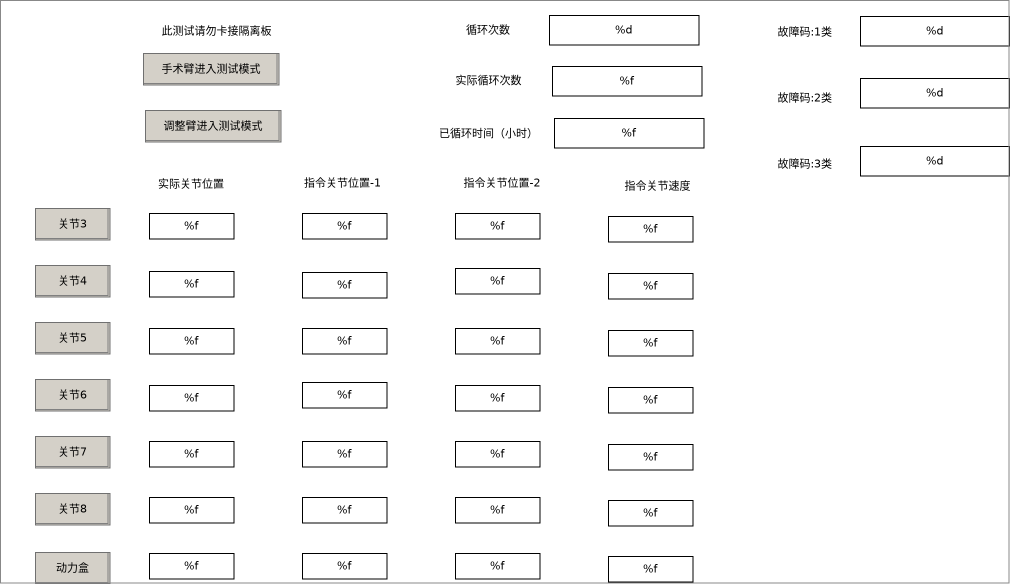
VISUALIZATION arm4CycleTest  // 1010x584
VAR_IN_OUT
	
END_VAR
VAR CONSTANT
	arm : INT := 4;
END_VAR
    Button (143,53 136x32), "手术臂进入测试模式", colour toggle: g_cycleTest.m_enterCycleTestMode[4]
        toggle g_cycleTest.m_enterCycleTestMode[4]
    Rectangle (549,15 150x30), "%d", text variable: g_cycleTest.m_targetCycleNum[4]
    Label (446,15 84x30), "循环次数"
    Label (283,169 119x28), "指令关节位置-1"
    Label (141,169 100x30), "实际关节位置"
    Rectangle (149,385 85x26), "%f", text variable: g_systemInfo.m_slaveJntInfo[4,1].m_curJntPos
    Rectangle (149,441 85x26), "%f", text variable: g_systemInfo.m_slaveJntInfo[4,2].m_curJntPos
    Rectangle (149,497 85x26), "%f", text variable: g_systemInfo.m_slaveJntInfo[4,3].m_curJntPos
    Rectangle (149,553 85x26), "%f", text variable: g_systemInfo.m_slaveJntInfo[4,4].m_curJntPos
    Rectangle (149,213 85x26), "%f", text variable: g_systemInfo.m_setupJntInfo[4,3].m_curJntPos
    Rectangle (149,271 85x26), "%f", text variable: g_systemInfo.m_setupJntInfo[4,4].m_curJntPos
    Rectangle (149,328 85x26), "%f", text variable: g_systemInfo.m_setupJntInfo[4,5].m_curJntPos
    Rectangle (302,213 85x26), "%f", text variable: g_cycleTest.m_targetJntPosSetup[4,1][3]
        OnMouseClick: write the text variable via Default
    Rectangle (302,272 85x26), "%f", text variable: g_cycleTest.m_targetJntPosSetup[4,1][4]
        OnMouseClick: write the text variable via Default
    Rectangle (302,328 85x26), "%f", text variable: g_cycleTest.m_targetJntPosSetup[4,1][5]
        OnMouseClick: write the text variable via Default
    Rectangle (302,382 85x26), "%f", text variable: g_cycleTest.m_targetJntPos[4,1][1]
        OnMouseClick: write the text variable via Default
    Rectangle (302,441 85x26), "%f", text variable: g_cycleTest.m_targetJntPos[4,1][2]
        OnMouseClick: write the text variable via Default
    Rectangle (302,497 85x26), "%f", text variable: g_cycleTest.m_targetJntPos[4,1][3]
        OnMouseClick: write the text variable via Default
    Rectangle (302,553 85x26), "%f", text variable: g_cycleTest.m_targetJntPos[4,1][4]
        OnMouseClick: write the text variable via Default
    Label (444,169 116x28), "指令关节位置-2"
    Rectangle (455,213 85x26), "%f", text variable: g_cycleTest.m_targetJntPosSetup[4,2][3]
        OnMouseClick: write the text variable via Default
    Rectangle (455,268 85x26), "%f", text variable: g_cycleTest.m_targetJntPosSetup[4,2][4]
        OnMouseClick: write the text variable via Default
    Rectangle (455,328 85x26), "%f", text variable: g_cycleTest.m_targetJntPosSetup[4,2][5]
        OnMouseClick: write the text variable via Default
    Rectangle (455,385 85x26), "%f", text variable: g_cycleTest.m_targetJntPos[4,2][1]
        OnMouseClick: write the text variable via Default
    Rectangle (455,441 85x26), "%f", text variable: g_cycleTest.m_targetJntPos[4,2][2]
        OnMouseClick: write the text variable via Default
    Rectangle (455,497 85x26), "%f", text variable: g_cycleTest.m_targetJntPos[4,2][3]
        OnMouseClick: write the text variable via Default
    Rectangle (455,553 85x26), "%f", text variable: g_cycleTest.m_targetJntPos[4,2][4]
        OnMouseClick: write the text variable via Default
    Button (145,110 136x32), "调整臂进入测试模式", colour toggle: g_cycleTest.m_enterCycleTestModeSetup[4]
        toggle g_cycleTest.m_enterCycleTestModeSetup[4]
    Label (603,172 109x28), "指令关节速度"
    Rectangle (608,216 85x26), "%f", text variable: g_cycleTest.m_targetJntVelSetup[4][3]
        OnMouseClick: write the text variable via Default
    Rectangle (608,273 85x26), "%f", text variable: g_cycleTest.m_targetJntVelSetup[4][4]
        OnMouseClick: write the text variable via Default
    Rectangle (608,330 85x26), "%f", text variable: g_cycleTest.m_targetJntVelSetup[4][5]
        OnMouseClick: write the text variable via Default
    Rectangle (608,387 85x26), "%f", text variable: g_cycleTest.m_targetJntVelSlave[4][1]
        OnMouseClick: write the text variable via Default
    Rectangle (608,444 85x26), "%f", text variable: g_cycleTest.m_targetJntVelSlave[4][2]
        OnMouseClick: write the text variable via Default
    Rectangle (608,500 85x26), "%f", text variable: g_cycleTest.m_targetJntVelSlave[4][3]
        OnMouseClick: write the text variable via Default
    Rectangle (608,556 85x26), "%f", text variable: g_cycleTest.m_targetJntVelSlave[4][4]
        OnMouseClick: write the text variable via Default
    Rectangle (552,66 150x30), "%f", text variable: g_cycleTest.m_curCycleNum[4]
        OnMouseClick: write the text variable via Default
    Label (440,70 97x21), "实际循环次数"
    Rectangle (554,118 150x30), "%f", text variable: g_cycleTest.m_curCycleTime[4]
        OnMouseClick: write the text variable via Default
    Label (428,123 121x21), "已循环时间（小时）"
    Rectangle (860,16 150x30), "%d", text variable: GVL_interactUI.g_errIdType1
        OnMouseClick: write the text variable via Default
    Label (764,17 82x30), "故障码:1类"
    Rectangle (860,78 150x30), "%d", text variable: GVL_interactUI.g_errIdType2
        OnMouseClick: write the text variable via Default
    Label (764,83 82x30), "故障码:2类"
    Rectangle (860,146 150x30), "%d", text variable: GVL_interactUI.g_errIdType3
        OnMouseClick: write the text variable via Default
    Label (764,149 82x30), "故障码:3类"
    Button (35,208 75x32), "关节3", colour toggle: g_cycleTest.m_disableSetupJntMotion[4][3]
        toggle g_cycleTest.m_disableSetupJntMotion[4][3]
    Button (35,265 75x32), "关节4", colour toggle: g_cycleTest.m_disableSetupJntMotion[4][4]
        toggle g_cycleTest.m_disableSetupJntMotion[4][4]
    Button (35,322 75x32), "关节5", colour toggle: g_cycleTest.m_disableSetupJntMotion[4][5]
        toggle g_cycleTest.m_disableSetupJntMotion[4][5]
    Button (35,379 75x32), "关节6", colour toggle: g_cycleTest.m_disableSlaveJntMotion[4][1]
        toggle g_cycleTest.m_disableSlaveJntMotion[4][1]
    Button (35,436 75x32), "关节7", colour toggle: g_cycleTest.m_disableSlaveJntMotion[4][2]
        toggle g_cycleTest.m_disableSlaveJntMotion[4][2]
    Button (35,493 75x32), "关节8", colour toggle: g_cycleTest.m_disableSlaveJntMotion[4][3]
        toggle g_cycleTest.m_disableSlaveJntMotion[4][3]
    Button (35,552 75x32), "动力盒", colour toggle: g_cycleTest.m_disableSlaveJntMotion[4][4]
        toggle g_cycleTest.m_disableSlaveJntMotion[4][4]
    Label (140,16 153x30), "此测试请勿卡接隔离板"
END_VISUALIZATION

(* stored: Version 1.1.0.1, ProductVersion 3.1.4024.11
   Visu arm4CycleTest: Id {1c1f2ae1-52fd-44e3-8559-746d8b71d94e} *)
